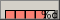
VISUALIZATION _VISU_CameraTrigger  // 60x20
VAR_IN_OUT
	mInst : FB_MarkDetection;
END_VAR
    RoundedRectangle (0,0 60x20), tooltip "Trigger Armed", colour toggle: mInst.bTriggerArmed
    RoundedRectangle (15,10 10x10), tooltip "Speed valid", colour toggle: mInst.bSpeedValid
    RoundedRectangle (25,10 10x10), tooltip "Cam valid", colour toggle: mInst.bCamValid
    RoundedRectangle (35,10 10x10), tooltip "(Hw)Enable", colour toggle: mInst.bEnable
    RoundedRectangle (5,10 10x10), tooltip "Init ok", colour toggle: mInst.bInitOk
    Rectangle (0,0 60x10), tooltip "Trigger active"
    RoundedRectangle (45,10 10x10), "%d", tooltip "e state", text variable: mInst.nMarkSelection
END_VISUALIZATION

(* stored: Version 1.1.0.1, ProductVersion 3.1.4024.11
   Visu _VISU_CameraTrigger: Id {224e6f8b-5cce-438f-8280-9a3f9ebd2872} *)
